PROGRAM Simulation
VAR
	rSpeed: REAL := 0;
	rPos: REAL := 0;
	bPulse: BOOL := TRUE;
	fbTon: TON;
END_VAR

fbTon(IN := NOT fbTon.Q, PT:= T#1S);
IF (fbTon.Q) THEN
	IF (rSpeed < 100) THEN
		rSpeed := rSpeed + 1.1;
	ELSE 
		rSpeed := 0;
	END_IF
	IF (rPos < 100) THEN
		rPos := rPos + 1;
	ELSE 
		rPos := 0;
	END_IF
	bPulse := NOT bPulse;
END_IF

END_PROGRAM

(* stored: Version 1.1.0.1, ProductVersion 3.1.4024.4
   POU Simulation: Id {f7d866ac-478f-42ea-9426-db5e34d2e00c}, SpecialFunc None *)
